INTERFACE ITF_Actuator_HMI_Connector EXTENDS ITF_BaseControlElement_HMI_Connector

METHOD GetTimeLastMove : TIME
VAR_INPUT
END_VAR
END_METHOD

METHOD IsEnd : BOOL
VAR_INPUT
END_VAR
END_METHOD

METHOD PUBLIC IsStart : BOOL
VAR_INPUT
END_VAR
END_METHOD

(*			
	EVERDE sp. z o.o.
	Rafał Osajda		31.03.2025		TC 4024.66
	Uruchomienie cyklu przesuwania do początku
*)
METHOD PUBLIC MoveToEnd
VAR_INPUT
END_VAR
END_METHOD

(*			
	EVERDE sp. z o.o.
	Rafał Osajda		31.03.2025		TC 4024.66
	Uruchomienie cyklu przesuwania do początku
*)
METHOD PUBLIC MoveToStart
VAR_INPUT
END_VAR
END_METHOD

METHOD PUBLIC MovingToEndBusy : BOOL
VAR_INPUT
END_VAR
END_METHOD

METHOD PUBLIC MovingToEndStatus : BOOL
VAR_INPUT
END_VAR
END_METHOD

METHOD PUBLIC MovingToStartBusy : BOOL
VAR_INPUT
END_VAR
END_METHOD

METHOD PUBLIC MovingToStartStatus : BOOL
VAR_INPUT
END_VAR
END_METHOD

END_INTERFACE

(* stored: Version 1.1.0.1
   Itf ITF_Actuator_HMI_Connector: Id {4e5d249e-46e7-4d89-9fee-0ce19c6739dc}
   Method GetTimeLastMove: Id {b6db5e0e-a9ec-458d-af33-d4b5180b6cf9}
   Method IsEnd: Id {ce93a036-1d75-4818-845b-9009db264e5f}
   Method IsStart: Id {5ea35caf-5189-4114-9423-26d426b8687c}
   Method MoveToEnd: Id {3006b99f-44e9-40f1-95c8-49a478cbb81b}
   Method MoveToStart: Id {908e00cc-d40c-427f-8007-88045ebc36fe}
   Method MovingToEndBusy: Id {5789098d-8fe2-4fa2-8dec-61be9c2c754c}
   Method MovingToEndStatus: Id {589ca5f2-a27e-4f30-be6e-32c194b1c5af}
   Method MovingToStartBusy: Id {fd3fd96c-73d8-40d1-ad72-f7545efc22d5}
   Method MovingToStartStatus: Id {4709a4ce-2684-41d9-b396-bdce4d01f751} *)
